Universal Robots PolyScope program: nastro 3binf.urp

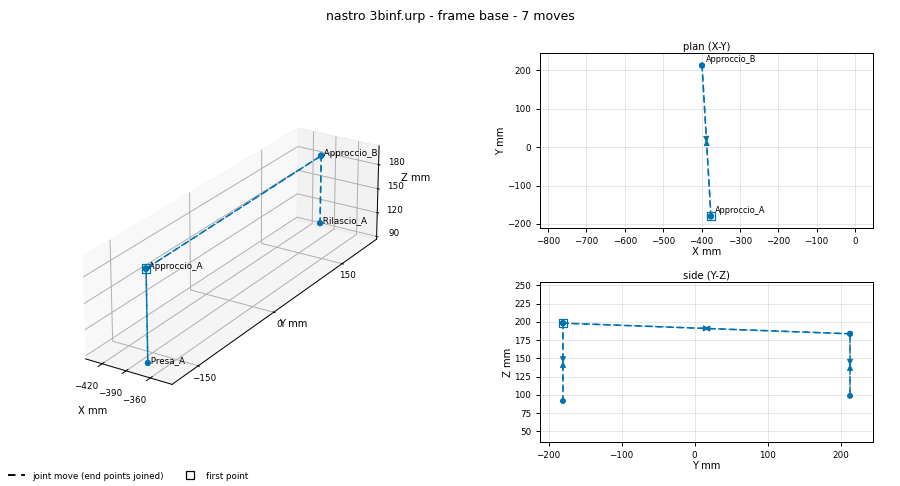
[picture p0: tool path of nastro 3binf.urp in frame base, 7 of 7 moves have a stored position in this frame; points joined in program order, loops and branches not executed]
Program nastro 3binf (installation=default directory=/programs createdIn=3.15.8.106339 lastSavedIn=3.15.8.106339 robotSerialNumber=2021330429)
Calibrated DH parameters: a=[-0.000156, -0.236402, -0.171625, 0.000006, -0.000047, 0]; d=[0.151683, 29.702709, 78.973085, -108.563557, 0.085229, 0.082167]; alpha=[1.57015, 0.001987, 0.001164, 1.571718, -1.571778, 0]; deltaTheta=[-0.000066, 0.24449, 0.39032, -0.635025, 0.000068, -0.000043]
BeforeStart
  Timer (action=Stop) variable(name=volo)
  ready := False
Robot Program (runOnlyOnce=false)
  Wait Condition expression=ready≟ True
  MoveJ speed 60 deg/s, acceleration 80 deg/s^2 (useActiveTCP=true)
    Waypoint Approccio_A: TCP in base x=-375.41 y=-180.261 z=198.07 mm, rx=-2.1145 ry=2.241 rz=0.0186 rad; joints [221.81, -123.705, -32.132, -117.533, 89.311, 225.041] deg; flange x=-381 y=-188.14 z=354.773 mm, rx=-2.1145 ry=2.241 rz=0.0186 rad
    Waypoint Presa_A: TCP in base x=-375.402 y=-180.303 z=91.469 mm, rx=-2.1146 ry=2.241 rz=0.0185 rad; joints [221.833, -119.109, -68.861, -85.398, 89.336, 225.081] deg; flange x=-380.997 y=-188.167 z=248.172 mm, rx=-2.1146 ry=2.241 rz=0.0185 rad
    URCap Gripper (Robotiq_Grippers, Robotiq Inc.) dataModel(position=100.0, force=0.0, speed=50.0, positionInDouble=100.0, forceInDouble=0.0, speedInDouble=50.0, slaveIds=[9], blocking=true)
    Waypoint Uscita_A: TCP in base x=-375.445 y=-180.236 z=198.105 mm, rx=-2.1146 ry=2.2412 rz=0.0186 rad; joints [221.805, -123.704, -32.127, -117.531, 89.31, 225.036] deg; flange x=-381.017 y=-188.102 z=354.808 mm, rx=-2.1146 ry=2.2412 rz=0.0186 rad
    Waypoint Approccio_B: TCP in base x=-398.72 y=212.86 z=183.511 mm, rx=-2.124 ry=2.3088 rz=-0.035 rad; joints [166.05, -133.687, -19.474, -117.972, 90.621, 170.711] deg; flange x=-401.577 y=214.996 z=340.471 mm, rx=-2.124 ry=2.3088 rz=-0.035 rad
    Waypoint Rilascio_A: TCP in base x=-398.747 y=212.833 z=98.51 mm, rx=-0.077 ry=-3.128 rz=0.0296 rad; joints [165.692, -124.959, -59.004, -85.517, 91.349, 258.428] deg; flange x=-396.717 y=215.758 z=255.47 mm, rx=-0.077 ry=-3.128 rz=0.0296 rad
    URCap Gripper (Robotiq_Grippers, Robotiq Inc.) dataModel(position=0.0, force=0.0, speed=50.0, positionInDouble=0.0, forceInDouble=0.0, speedInDouble=50.0, slaveIds=[9], blocking=true)
    Waypoint Approccio_B: TCP in base x=-398.72 y=212.86 z=183.511 mm, rx=-2.124 ry=2.3088 rz=-0.035 rad; joints [166.05, -133.687, -19.474, -117.972, 90.621, 170.711] deg; flange x=-401.577 y=214.996 z=340.471 mm, rx=-2.124 ry=2.3088 rz=-0.035 rad
    Waypoint Approccio_A: TCP in base x=-375.41 y=-180.261 z=198.07 mm, rx=-2.1145 ry=2.241 rz=0.0186 rad; joints [221.81, -123.705, -32.132, -117.533, 89.311, 225.041] deg; flange x=-381 y=-188.14 z=354.773 mm, rx=-2.1145 ry=2.241 rz=0.0186 rad
Thread Thread_1 (runOnlyOnce=false)
  If digital_in[6]≟ True
    Timer (action=Stop) variable=volo
    Set DigitalOutput pin=digital_out[0]; digitalValue=1
    Wait DigitalInput pin=digital_in[6]; digitalValue=0
  ElseIf digital_in[4]≟ True
    Timer (action=Stop) variable=volo
    Set DigitalOutput pin=digital_out[0]; digitalValue=1
    Wait DigitalInput pin=digital_in[5]; digitalValue=0
  ElseIf digital_in[5]≟ True
    Timer (action=Stop) variable=volo
    Timer (action=Reset) variable=volo
    Wait Sleep waitTime=0.5
    Set DigitalOutput pin=digital_out[0]; digitalValue=0
    ready := True
    Wait DigitalInput pin=digital_in[5]; digitalValue=0
    ready := False
    Set DigitalOutput pin=digital_out[0]; digitalValue=1
    Timer (action=Start) variable=volo
  If volo≥10
    Set DigitalOutput pin=digital_out[0]; digitalValue=0
    Timer (action=Reset) variable=volo
    Timer (action=Stop) variable=volo
